(****************************************************************************************)
(*							Beckhoff Automation Poland									*)
(*								FB_IntTo2Byte	 v1.0									*)
(*									24.5.2011											*)
(*			Blok funkcyjny rozbijający zmienną typu INT na dwie zmienne typu BYTE		*)
(*______________________________________________________________________________________*)
FUNCTION_BLOCK FB_IntTo2Byte
VAR_INPUT
	iInput :INT;
END_VAR
VAR_OUTPUT
	byStarszy : BYTE;
	byMlodszy : BYTE;
END_VAR

byMlodszy := INT_TO_BYTE(iInput);
byStarszy := INT_TO_BYTE(ROL(iInput, 8));

END_FUNCTION_BLOCK

(* stored: Version 1.1.0.1, ProductVersion 3.1.4026.13, FileIdentifier 0767569121dee07e2377a0368d70433b4ba1dac7, FileSignature 907e0e9599db33528091dc48d86a2dded08ba9b3fa8e0680d008e3c04be093e992b06be8662bd02d965fcb547093b8a4890fae90f19edeeccc99aa0b9cc4e5aab0f757798ef8352ddff7458fd49e535f06fbdac279501837f2bab3745571c094ad4168f97681a4e9dffca9af8d7092abb0d94320f7759aadff6a81bfc065831e9af44840d3173eab6929c67c7d6e1cc3862ce6fb137ad443f66eb997f83c82a7a1e82cf38c466117be248cf7a1103bc202676fc32b0911c2c5edb6a561fb54b5e5dabd0ba1e3ea0e03eda28374974cbaac375a2d8b8c5227a491a8b2c4cc10f772a2dbb76caa80c895a60a2c385d5f346ca905cf88cadb2ed594c084a7d9f795
   POU FB_IntTo2Byte: Id {7e7a398c-7c24-4d3f-96a5-6db969f8671e}, SpecialFunc None *)
